// TIA Portal V20 export
TYPE "typeAxisJogCondition"
// stored: Access Published, Namespace LER
   STRUCT
      ForwardInterlockOK : Bool;
      BackwardInterlockOk : Bool;
      ForwardInterlockError : Bool;
      BackwardInterlockError : Bool;
      intOut : Array[0..9] of Bool;
   END_STRUCT;
END_TYPE
